{attribute 'qualified_only'}
VAR_GLOBAL CONSTANT
(* Star Wars Imperial March *) 
	Beeps : ARRAY[0..201] OF REAL := [392, 350, 100, 392, 350, 100, 392, 350, 100, 311, 250, 100, 466, 25, 100, 392, 350, 100, 311, 250, 100, 466, 25, 100, 392, 700, 100, 587, 350, 100, 587, 350, 100, 587, 350, 100, 622, 250, 100, 466, 25, 100, 369, 350, 100, 311, 250, 100, 466, 25, 100, 392, 700, 100, 784, 350, 100, 392, 250, 100, 392, 25, 100, 784, 350, 100, 739, 250, 100, 698, 25, 100, 659, 25, 100, 622, 25, 100, 659, 50, 400, 415, 25, 200, 554, 350, 100, 523, 250, 100, 493, 25, 100, 466, 25, 100, 440, 25, 100, 466, 50, 400, 311, 25, 200, 369, 350, 100, 311, 250, 100, 392, 25, 100, 466, 350, 100, 392, 250, 100, 466, 25, 100, 587, 700, 100, 784, 350, 100, 392, 250, 100, 392, 25, 100, 784, 350, 100, 739, 250, 100, 698, 25, 100, 659, 25, 100, 622, 25, 100, 659, 50, 400, 415, 25, 200, 554, 350, 100, 523, 250, 100, 493, 25, 100, 466, 25, 100, 440, 25, 100, 466, 50, 400, 311, 25, 200, 392, 350, 100, 311, 250, 100, 466, 25, 100, 392, 300, 150, 311, 250, 100, 466, 25, 100, 392, 700, 0, 0, 0, 0];
END_VAR

(* stored: Version 1.1.0.1, ProductVersion 3.1.4019.2
   GVL StarWars: Id {9de6ecac-470f-47be-b10f-9bd31bd006c7} *)
